{attribute 'GeneratedUsingTerminal: EK1100-0000-0018'}
{attribute addProperty BoxType "EK1100-0000-0018"}
{attribute addProperty Id "Beckhoff_EP2xxxEK1122Beckhoff_EP2xxxEK1122_6A4FE0FF3524"}
{attribute addProperty CRC "1584121181"}
{attribute addProperty Size "3524"}
{attribute addProperty Name "Beckhoff EP2xxx"}
TYPE Beckhoff_EP2xxx_5E6BC55D EXTENDS EK1100_1FC0878B :
STRUCT
	{attribute addProperty Name "Beckhoff EP2xxxEK1122"}
	{attribute addProperty PreviousPort "Beckhoff EP2xxx : B"}
	Beckhoff_EP2xxxEK1122 : Beckhoff_EP2xxxEK1122_6A4FE0FF;
END_STRUCT
END_TYPE

(* stored: Version 1.2.0.0, ProductVersion 3.1.4024.11
   DUT Beckhoff_EP2xxx_5E6BC55D: Id {ab36cff6-46c6-42da-8f49-97704cbd3693} *)
